INTERFACE I_LinearContinuousDrive EXTENDS I_LinearDrive, I_ContinuousDrive

END_INTERFACE

(* stored: Version 1.1.0.1, ProductVersion 3.1.4024.11
   Itf I_LinearContinuousDrive: Id {de988ca7-8253-4553-b5c2-9396bb5bd9b0} *)
